// Mitsubishi GX Works2 project: q6   PLC: Q02/Q02H

PROGRAM MAIN
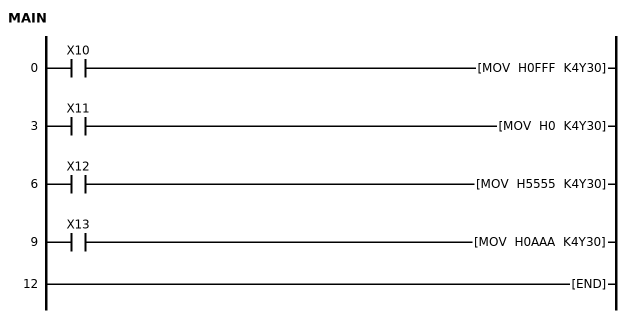
0     LD      X10
      MOV     H0FFF K4Y30
3     LD      X11
      MOV     H0 K4Y30
6     LD      X12
      MOV     H5555 K4Y30
9     LD      X13
      MOV     H0AAA K4Y30
12    END
END_PROGRAM
